//project related global variables
{attribute 'qualified_only'}
{attribute 'analysis' := '-33'}
VAR_GLOBAL
//Checkbounds can be disabled by setting exclude from build is true at the properties of this block
//NOTE: getting it on again, can be a bit of a hassle, 
//	-include checkbounds in build
//  -add some variable to this global struct >> now this will get rebuild with the variables needed for checkbounds
{IF defined (pou: CHECKBOUNDS)}
	{warning 'CHECKBOUNDS is active, this causes increased processor load. Exclude block from build when possible'}
	OutOfBounds:BOOL:=FALSE;						//Should always be false otherwise a bounds problem >> function CHECKBOUNDS must be implemented in the project, check the beckhoff help !only for testing purposes!
	OutOfBoundsIndex:DINT := 0;						//Index trying to address which was out of bounds
{END_IF}

(*Project*)
	Sim_MyMachinePart:BOOL; //only here as example, remove me
	Sim_WithoutSql:BOOL;
END_VAR
// {attribute 'qualified_only'} >>forces the user to add the DUT name in front of the variables
// {attribute 'analysis' := '-33'} >>deactivate error unused variable for next variable/struct

(* stored: Version 1.1.0.1, ProductVersion 3.1.4024.12
   GVL Glbl: Id {c945def9-01c5-4958-81b0-c5c4c71d8d05} *)
